{attribute addProperty BoxType "EP7402-0057-0017"}
{attribute addProperty Id "Device_DiagAT %I*Device_Diag_EB02919D324"}
{attribute addProperty CRC "2590067136"}
{attribute addProperty SizeInBites "32"}
{attribute addProperty SizeInBytes "4"}
TYPE STM_Inputs_Device_9A6149C0 :
STRUCT
	{attribute addProperty Name "Device_Diag"}
	Device_Diag AT %I* : Device_Diag_EB02919D;
END_STRUCT
END_TYPE

(* stored: Version 1.2.0.0, ProductVersion 3.1.4024.9
   DUT STM_Inputs_Device_9A6149C0: Id {afd58664-46e2-4460-8abe-3e3c074abce5} *)
